(* PLC project Math Expression Evaluator, CODESYS CODESYS V3.5 SP18 Patch 5 *)
(* stored: creationDateTime 2024-02-04T11:49:45.7079355, version 0.1.0.0, modificationDateTime 2024-02-04T11:49:30.3793356, organization GG *)
(* The Math Expression Evaluator evaluates math expressions (terms).

See the documentation folder for an introduction (the folder itself). *)

TYPE typExpressionStep : STRUCT
  atTokens : ARRAY[0..ParameterList.uiMaxExpressionTokens] OF typExpressionToken;
  uiCountTokens : UINT;
  uiInternalVariableTarget : UINT;
END_STRUCT;
END_TYPE

TYPE typExpressionToken : STRUCT
  eType : eTokenType;
  uiGroupNumber : UINT;
  sIdentifier : STRING(5);
  uiArgsCount : UINT;
  xArgsVariable : BOOL;
  lrValue : LREAL;
END_STRUCT;
END_TYPE

TYPE typStepizeGroupFound : STRUCT
  uiTokenIndex : UINT;
  uiGroupNumber : UINT;
  xExpandMore : BOOL;
END_STRUCT;
END_TYPE

TYPE typStepizeRewriteTokenSkips : STRUCT
  uiStart : UINT;
  uiEnd : UINT;
  uiVarNum : UINT;
END_STRUCT;
END_TYPE

(* A division by zero is not allowed and this ENUM describes how such a situation is handled. - ERROR: An error is returned - RESULT_IS_ZERO: The result is simply set to 0.0 and no error is returned - DIVISOR_IS_ONE: The divisor is set to 1.0 instead and the operation is being carried out *)
{attribute 'qualified_only'}
{attribute 'strict'}
TYPE eDivisionByZeroHandling : (ERROR := 0, RESULT_IS_ZERO, DIVISOR_IS_ONE);
END_TYPE

{attribute 'qualified_only'}
{attribute 'strict'}
TYPE eTokenType : (INVALID := 0, NUMBER, VARIABLE, GROUP_START, GROUP_END, MATH_OP, FUNCTION_CALL, FUNCTION_CALL_END, INTERNAL_VAR := 99);
END_TYPE

TYPE typExpressionOperationSteps : STRUCT
  atSteps : ARRAY[0..ParameterList.uiMaxStepsPerOperation] OF typExpressionStep;
  uiCountSteps : UINT;
END_STRUCT;
END_TYPE

TYPE typTokenizedExpression : STRUCT
  atTokens : ARRAY[0..ParameterList.uiMaxExpressionTokens] OF typExpressionToken;
  uiCountTokens : UINT;
END_STRUCT;
END_TYPE

{attribute 'qualified_only'}
VAR_GLOBAL CONSTANT  (* Constants *)
  CHAR_WHITESPACE : BYTE := 32;
  CHAR_NEWLINE : BYTE := 10;
  CHAR_CAR_RETURN : BYTE := 13;
  CHAR_VARIABLE : BYTE := 92;  (* \ *)
  CHAR_GROUP_START : BYTE := 40;  (* ( *)
  CHAR_GROUP_END : BYTE := 41;  (* ) *)
  CHAR_COMMA : BYTE := 44;  (* , *)
  CHAR_DOT : BYTE := 46;  (* . *)
  CHAR_LC_E : BYTE := 101;  (* e *)
  CHAR_ADD : BYTE := 43;  (* + (also used for sign) *)
  CHAR_SUB : BYTE := 45;  (* - (also used for sign) *)
  CHAR_MUL : BYTE := 42;  (* * *)
  CHAR_DIV : BYTE := 47;  (* / *)
  CHAR_EXP : BYTE := 94;  (* ^ *)
  CHAR_MOD : BYTE := 37;  (* % *)
  ASCII_ALPHA_START : BYTE := 65;  (* A *)
  ASCII_ALPHA_END : BYTE := 90;  (* Z *)
  ASCII_NUM_START : BYTE := 48;  (* 0 *)
  ASCII_NUM_END : BYTE := 57;  (* 9 *)
  MAX_FUN_ARGS : UINT := 9;
  FUN_ABS : STRING(5) := 'ABS';  (* Single arg functions *)
  FUN_ACOS : STRING(5) := 'ACOS';
  FUN_ASIN : STRING(5) := 'ASIN';
  FUN_ATAN : STRING(5) := 'ATAN';
  FUN_CEIL : STRING(5) := 'CEIL';
  FUN_COS : STRING(5) := 'COS';
  FUN_DEG : STRING(5) := 'DEG';
  FUN_FLOOR : STRING(5) := 'FLOOR';
  FUN_LOG : STRING(5) := 'LOG';
  FUN_LN : STRING(5) := 'LN';
  FUN_RAD : STRING(5) := 'RAD';
  FUN_ROUND : STRING(5) := 'ROUND';
  FUN_SIN : STRING(5) := 'SIN';
  FUN_SQRT : STRING(5) := 'SQRT';
  FUN_TAN : STRING(5) := 'TAN';
  FUN_TRUNC : STRING(5) := 'TRUNC';  (* Dual arg functions *)
  FUN_LIMIT : STRING(5) := 'LIMIT';  (* Triple arg functions *)
  FUN_AVGA : STRING(5) := 'AVG';  (* Variable arg functions (2..9) *)
  FUN_MAX : STRING(5) := 'MAX';
  FUN_MIN : STRING(5) := 'MIN';
END_VAR

{attribute 'parameterlist'}
{attribute 'qualified_only'}
VAR_GLOBAL CONSTANT  (* ParameterList *)
  uiMaxExpressionTokens : UINT := 63;  (* The maximum amount of tokens to support parsing (compiling) - the counting starts from 0, so add 1 to the number in your mind *)
  uiMaxInternalVars : UINT := 16;  (* The maximum amount of internal variables per expression *)
  uiMaxStepsPerOperation : UINT := 15;  (* The maximum amount of steps per operation - the counting starts from 0, so add 1 to the number in your mind *)
  eDivisionByZero : eDivisionByZeroHandling := eDivisionByZeroHandling.ERROR;  (* Describes how a division by zero situation is to be handled *)
END_VAR

(* Evaluates a function call. First all necessary arguments are resolved to LREAL and then the function gets executed. The return value will indicate a successful evaluation. *)
{attribute 'qualified_only'}
FUNCTION FuEvaluateFunctionCall : BOOL
  VAR_INPUT
    typFunctionToken : typExpressionToken;
    uiMaxCursor : UINT;
    {attribute 'variable_length_array_original_scope' := 'Inout'}
    {attribute 'variable_length_array' := 'ARRAY[*] OF typExpressionToken'}
    {attribute 'Dimensions' := '1'}
    atTokens : POINTER TO typExpressionToken;
  END_VAR
  VAR_IN_OUT
    uiCursor : UINT;
  END_VAR
  VAR_INPUT
    {attribute 'variable_length_array_original_scope' := 'Inout'}
    {attribute 'variable_length_array' := 'ARRAY[*] OF LREAL'}
    {attribute 'Dimensions' := '1'}
    alrVariables : POINTER TO LREAL;
    {attribute 'variable_length_array_original_scope' := 'Inout'}
    {attribute 'variable_length_array' := 'ARRAY[*] OF LREAL'}
    {attribute 'Dimensions' := '1'}
    alrInternalVariables : POINTER TO LREAL;
  END_VAR
  VAR_OUTPUT
    lrResult : LREAL;
    sError : STRING;
  END_VAR
  VAR
    i : UINT;
    j : UINT;
    tempArgs : ARRAY[0..8] OF LREAL;
    tempHelperValue : LREAL;
  END_VAR
  VAR CONSTANT
    CONST_PI : LREAL := 3.14159265359;
  END_VAR

            IF typFunctionToken.eType <> eTokenType.FUNCTION_CALL THEN
    sError := Standard.CONCAT('Invalid function call token at ', TO_STRING(uiCursor));
    RETURN;
END_IF

IF uiCursor + typFunctionToken.uiArgsCount > uiMaxCursor THEN
    sError := Standard.CONCAT('Not enough arguments for function call at ', TO_STRING(uiCursor));
    RETURN;
END_IF

FOR i := 0 TO (typFunctionToken.uiArgsCount - 1) BY 1 DO
    j := uiCursor + i + 1;
    
    IF NOT FuEvaluateTokenSingle(atTokens[j], j, alrVariables, alrInternalVariables, lrResult => tempArgs[i], sError => sError) THEN
        RETURN;
    END_IF
END_FOR

uiCursor := uiCursor + typFunctionToken.uiArgsCount;

IF typFunctionToken.sIdentifier = Constants.FUN_ABS THEN
    FuEvaluateFunctionCall := TRUE;
    lrResult := ABS(tempArgs[0]);
ELSIF typFunctionToken.sIdentifier = Constants.FUN_ACOS THEN
    FuEvaluateFunctionCall := TRUE;
    lrResult := ACOS(tempArgs[0]);
ELSIF typFunctionToken.sIdentifier = Constants.FUN_ASIN THEN
    FuEvaluateFunctionCall := TRUE;
    lrResult := ASIN(tempArgs[0]);
ELSIF typFunctionToken.sIdentifier = Constants.FUN_ATAN THEN
    FuEvaluateFunctionCall := TRUE;
    lrResult := ATAN(tempArgs[0]);
ELSIF typFunctionToken.sIdentifier = Constants.FUN_CEIL THEN
    FuEvaluateFunctionCall := TRUE;
    lrResult := FPU.Ceil(tempArgs[0]);
ELSIF typFunctionToken.sIdentifier = Constants.FUN_COS THEN
    FuEvaluateFunctionCall := TRUE;
    lrResult := COS(tempArgs[0]);
ELSIF typFunctionToken.sIdentifier = Constants.FUN_DEG THEN
    FuEvaluateFunctionCall := TRUE;
    lrResult := tempArgs[0] * 180 / CONST_PI;
ELSIF typFunctionToken.sIdentifier = Constants.FUN_FLOOR THEN
    FuEvaluateFunctionCall := TRUE;
    lrResult := FPU.Floor(tempArgs[0]);
ELSIF typFunctionToken.sIdentifier = Constants.FUN_LOG THEN
    FuEvaluateFunctionCall := TRUE;
    lrResult := LOG(tempArgs[0]);
ELSIF typFunctionToken.sIdentifier = Constants.FUN_LN THEN
    FuEvaluateFunctionCall := TRUE;
    lrResult := LN(tempArgs[0]);
ELSIF typFunctionToken.sIdentifier = Constants.FUN_RAD THEN
    FuEvaluateFunctionCall := TRUE;
    lrResult := tempArgs[0] * CONST_PI / 180;
ELSIF typFunctionToken.sIdentifier = Constants.FUN_ROUND THEN
    FuEvaluateFunctionCall := TRUE;
    
    IF (tempArgs[0] - FPU.Truncate(tempArgs[0])) >= 0.5 THEN
        lrResult := FPU.Ceil(tempArgs[0]);
    ELSE
        lrResult := FPU.Floor(tempArgs[0]);
    END_IF
ELSIF typFunctionToken.sIdentifier = Constants.FUN_SIN THEN
    FuEvaluateFunctionCall := TRUE;
    lrResult := SIN(tempArgs[0]);
ELSIF typFunctionToken.sIdentifier = Constants.FUN_SQRT THEN
    FuEvaluateFunctionCall := TRUE;
    lrResult := SQRT(tempArgs[0]);
ELSIF typFunctionToken.sIdentifier = Constants.FUN_TAN THEN
    FuEvaluateFunctionCall := TRUE;
    lrResult := TAN(tempArgs[0]);
ELSIF typFunctionToken.sIdentifier = Constants.FUN_TRUNC THEN
    FuEvaluateFunctionCall := TRUE;
    
    tempHelperValue := EXPT(10, tempArgs[1]);
    lrResult := FPU.Truncate((tempArgs[0] * tempHelperValue)) / tempHelperValue;
ELSIF typFunctionToken.sIdentifier = Constants.FUN_LIMIT THEN
    FuEvaluateFunctionCall := TRUE;
    lrResult := LIMIT(tempArgs[0], tempArgs[1], tempArgs[2]);
ELSIF typFunctionToken.sIdentifier = Constants.FUN_AVGA THEN
    FuEvaluateFunctionCall := TRUE;
    
    tempHelperValue := 0.0;
    FOR i := 0 TO (typFunctionToken.uiArgsCount - 1) BY 1 DO
        tempHelperValue := tempHelperValue + tempArgs[i];
    END_FOR
    
    lrResult := tempHelperValue / typFunctionToken.uiArgsCount;
ELSIF typFunctionToken.sIdentifier = Constants.FUN_MAX THEN
    FuEvaluateFunctionCall := TRUE;
    
    lrResult := -1.7976931348623157E+308;
    FOR i := 0 TO (typFunctionToken.uiArgsCount - 1) BY 1 DO
        IF tempArgs[i] > lrResult THEN
            lrResult := tempArgs[i];
        END_IF
    END_FOR
ELSIF typFunctionToken.sIdentifier = Constants.FUN_MIN THEN
    FuEvaluateFunctionCall := TRUE;
    
    lrResult := 1.7976931348623157E+308;
    FOR i := 0 TO (typFunctionToken.uiArgsCount - 1) BY 1 DO
        IF tempArgs[i] < lrResult THEN
            lrResult := tempArgs[i];
        END_IF
    END_FOR
ELSE
    sError := Standard.CONCAT('Function not implemented: ', typFunctionToken.sIdentifier);
END_IF

          
END_FUNCTION

(* Evaluates a math operation. First both tokens are resolved to LREAL values and then the selected operation takes place. In general, if any of the operands is a special LREAL value, then an error is returned. For Division (/), division by zero yields into an error (depends on ParameterList setting). For MODULO (%), both tokens are converted to LINT and the result is converted back to LREAL. The return value will indicate a successful evaluation. *)
{attribute 'qualified_only'}
FUNCTION FuEvaluateMathOp : BOOL
  VAR_INPUT
    typOp : typExpressionToken;
    typToken1 : typExpressionToken;
    typToken2 : typExpressionToken;
    uiCursor : UINT;  (* Only for error message *)
    {attribute 'variable_length_array_original_scope' := 'Inout'}
    {attribute 'variable_length_array' := 'ARRAY[*] OF LREAL'}
    {attribute 'Dimensions' := '1'}
    alrVariables : POINTER TO LREAL;
    {attribute 'variable_length_array_original_scope' := 'Inout'}
    {attribute 'variable_length_array' := 'ARRAY[*] OF LREAL'}
    {attribute 'Dimensions' := '1'}
    alrInternalVariables : POINTER TO LREAL;
  END_VAR
  VAR_OUTPUT
    lrResult : LREAL;
    sError : STRING;
  END_VAR
  VAR
    tempOperatorByte : BYTE;
    tempNumber1 : LREAL;
    tempNumber2 : LREAL;
  END_VAR

            IF typOp.eType <> eTokenType.MATH_OP THEN
    sError := Standard.CONCAT('Invalid math operation token at ', TO_STRING(uiCursor));
    RETURN;
END_IF

// Change STRING identifier to BYTE (to match on FuTokenizeExpression strings)
tempOperatorByte := typOp.sIdentifier[0];

// Resolve first token to LREAL
IF NOT FuEvaluateTokenSingle(typToken1, uiCursor, alrVariables, alrInternalVariables, lrResult => tempNumber1, sError => sError) THEN
    FuEvaluateMathOp := FALSE;
    RETURN;
END_IF

// Resolve second token to LREAL
IF NOT FuEvaluateTokenSingle(typToken2, uiCursor, alrVariables, alrInternalVariables, lrResult => tempNumber2, sError => sError) THEN
    FuEvaluateMathOp := FALSE;
    RETURN;
END_IF

IF NOT FPU.IsLRealNumber(tempNumber1) THEN
    FuEvaluateMathOp := FALSE;
    sError := Standard.CONCAT('Special LREAL value is not valid: ', TO_STRING(tempNumber1));
    RETURN;
ELSIF NOT FPU.IsLRealNumber(tempNumber2) THEN
    FuEvaluateMathOp := FALSE;
    sError := Standard.CONCAT('Special LREAL value is not valid: ', TO_STRING(tempNumber2));
    RETURN;
END_IF

IF tempOperatorByte = Constants.CHAR_ADD THEN
    lrResult := tempNumber1 + tempNumber2;
ELSIF tempOperatorByte = Constants.CHAR_SUB THEN
    lrResult := tempNumber1 - tempNumber2;
ELSIF tempOperatorByte = Constants.CHAR_MUL THEN
    lrResult := tempNumber1 * tempNumber2;
ELSIF tempOperatorByte = Constants.CHAR_DIV THEN
    IF tempNumber2 = 0.0 THEN
        CASE ParameterList.eDivisionByZero OF
            eDivisionByZeroHandling.RESULT_IS_ZERO:
                FuEvaluateMathOp := TRUE;
                lrResult := 0.0;
                RETURN;
            
            eDivisionByZeroHandling.DIVISOR_IS_ONE:
                tempNumber2 := 1.0;
        ELSE
            sError := 'Division by zero is not allowed';
            RETURN;
        END_CASE
    END_IF
    
    lrResult := tempNumber1 / tempNumber2;
ELSIF tempOperatorByte = Constants.CHAR_EXP THEN
    lrResult := EXPT(tempNumber1, tempNumber2);
ELSIF tempOperatorByte = Constants.CHAR_MOD THEN
    lrResult := LINT_TO_LREAL((LREAL_TO_LINT(tempNumber1) MOD LREAL_TO_LINT(tempNumber2)));
ELSE
    sError := Standard.CONCAT('Unknown math operator at position ', TO_STRING(uiCursor));
    RETURN;
END_IF

FuEvaluateMathOp := TRUE;

          
END_FUNCTION

(* Evaluates an operation expression. For example "5 + 2", but not "5 + 2 + 1". The return value will indicate a successful evaluation. *)
{attribute 'qualified_only'}
FUNCTION FuEvaluateOperation : BOOL
  VAR_INPUT
    uiMaxCursor : UINT;
    {attribute 'variable_length_array_original_scope' := 'Inout'}
    {attribute 'variable_length_array' := 'ARRAY[*] OF typExpressionToken'}
    {attribute 'Dimensions' := '1'}
    atTokens : POINTER TO typExpressionToken;
  END_VAR
  VAR_IN_OUT
    uiCursor : UINT;
  END_VAR
  VAR_INPUT
    {attribute 'variable_length_array_original_scope' := 'Inout'}
    {attribute 'variable_length_array' := 'ARRAY[*] OF LREAL'}
    {attribute 'Dimensions' := '1'}
    alrVariables : POINTER TO LREAL;
    {attribute 'variable_length_array_original_scope' := 'Inout'}
    {attribute 'variable_length_array' := 'ARRAY[*] OF LREAL'}
    {attribute 'Dimensions' := '1'}
    alrInternalVariables : POINTER TO LREAL;
  END_VAR
  VAR_OUTPUT
    lrResult : LREAL;
    sError : STRING;
  END_VAR
  VAR
    tempLowerBound : UINT;
    tempUpperBound : UINT;
    tempToken1 : typExpressionToken;
    tempToken2 : typExpressionToken;
    tempToken3 : typExpressionToken;
    tempVariableNr : UINT;
  END_VAR

            tempLowerBound := TO_UINT(LOWER_BOUND(atTokens, 1));
tempUpperBound := MIN(uiMaxCursor, TO_UINT(UPPER_BOUND(atTokens, 1)));

tempToken1 := atTokens[uiCursor];

CASE tempToken1.eType OF
    eTokenType.INVALID, eTokenType.MATH_OP, eTokenType.GROUP_START, eTokenType.GROUP_END, eTokenType.FUNCTION_CALL_END:
        sError := Standard.CONCAT('Invalid token at position ', TO_STRING(uiCursor));
        RETURN;
    
    eTokenType.FUNCTION_CALL:
        FuEvaluateOperation := FuEvaluateFunctionCall(
            tempToken1,
            tempUpperBound,
            atTokens,
            uiCursor,
            alrVariables,
            alrInternalVariables,
            lrResult => lrResult,
            sError => sError
        );
        RETURN;
END_CASE

// If we're past the maximum position/cursor, evaluate the token (it should be a variable or number)
IF uiCursor = uiMaxCursor AND_THEN FuEvaluateTokenSingle(tempToken1, uiCursor, alrVariables, alrInternalVariables, lrResult => lrResult, sError => sError) THEN
    RETURN;
END_IF

uiCursor := uiCursor + 1;

// The first token wasn't a variable or number and we're out of bounds, error out
IF uiCursor > tempUpperBound THEN
    sError := 'Array upper bounds violation (not enough tokens)';
    RETURN;
END_IF

tempToken2 := atTokens[uiCursor];

CASE tempToken2.eType OF
    eTokenType.MATH_OP:
        uiCursor := uiCursor + 1;
        IF uiCursor > tempUpperBound THEN
            sError := 'Array upper bounds violation (not enough tokens)';
            RETURN;
        END_IF
        
        FuEvaluateOperation := FuEvaluateMathOp(
            tempToken2,
            tempToken1,
            atTokens[uiCursor],
            uiCursor,
            alrVariables,
            alrInternalVariables,
            lrResult => lrResult,
            sError => sError
        );
        RETURN;
ELSE
    sError := Standard.CONCAT('Invalid token at position ', TO_STRING(uiCursor));
    RETURN;
END_CASE

          
END_FUNCTION

(* Evaluates a single step. For multiple token "expressions" (i.e. "5 + 2 + 1"), the term will be evaluated left to right (in token order). The return value will indicate a successful expression evaluation. *)
{attribute 'qualified_only'}
FUNCTION FuEvaluateStep : BOOL
  VAR_INPUT
    typStep : typExpressionStep;
  END_VAR
  VAR_OUTPUT
    lrResult : LREAL;
    sError : STRING;
  END_VAR
  VAR_INPUT
    {attribute 'variable_length_array_original_scope' := 'Inout'}
    {attribute 'variable_length_array' := 'ARRAY[*] OF LREAL'}
    {attribute 'Dimensions' := '1'}
    alrVariables : POINTER TO LREAL;
    {attribute 'variable_length_array_original_scope' := 'Inout'}
    {attribute 'variable_length_array' := 'ARRAY[*] OF LREAL'}
    {attribute 'Dimensions' := '1'}
    alrInternalVariables : POINTER TO LREAL;
  END_VAR
  VAR
    i : UINT;
    tempMaxCursor : UINT;
    tempResult : LREAL;
    tempError : STRING;
  END_VAR

            IF typStep.uiCountTokens = 0 THEN
    FuEvaluateStep := TRUE;
    RETURN;
END_IF

lrResult := 0.0;
sError := '';

tempMaxCursor := typStep.uiCountTokens - 1;
FOR i := 0 TO tempMaxCursor BY 1 DO
    // For operations like "5 + 3 + 1", we need for the second step "+ 1"
    // to insert the previous result of "5 + 3", so we rewind one and overwrite it
    IF i > 0 AND_THEN typStep.atTokens[i].eType = eTokenType.MATH_OP THEN
        i := i - 1;
        typStep.atTokens[i].eType := eTokenType.NUMBER;
        typStep.atTokens[i].lrValue := tempResult;
    END_IF
    
    IF NOT FuEvaluateOperation(tempMaxCursor, typStep.atTokens, i, alrVariables, alrInternalVariables, lrResult => tempResult, sError => tempError) THEN
        sError := tempError;
        RETURN;
    END_IF
END_FOR

lrResult := tempResult;
FuEvaluateStep := TRUE;

          
END_FUNCTION

(* Evaluates token types that are considered "single". This includes: numbers, variables, internal variables. The return value will indicate a successful evaluation. *)
{attribute 'qualified_only'}
FUNCTION FuEvaluateTokenSingle : BOOL
  VAR_INPUT
    typToken : typExpressionToken;
    uiCursor : UINT;  (* Only for error message *)
    {attribute 'variable_length_array_original_scope' := 'Inout'}
    {attribute 'variable_length_array' := 'ARRAY[*] OF LREAL'}
    {attribute 'Dimensions' := '1'}
    alrVariables : POINTER TO LREAL;
    {attribute 'variable_length_array_original_scope' := 'Inout'}
    {attribute 'variable_length_array' := 'ARRAY[*] OF LREAL'}
    {attribute 'Dimensions' := '1'}
    alrInternalVariables : POINTER TO LREAL;
  END_VAR
  VAR_OUTPUT
    lrResult : LREAL;
    sError : STRING;
  END_VAR
  VAR
    tempVariableNr : UINT;
  END_VAR

            CASE typToken.eType OF
    eTokenType.NUMBER:
        FuEvaluateTokenSingle := TRUE;
        lrResult := typToken.lrValue;
    
    eTokenType.VARIABLE, eTokenType.INTERNAL_VAR:
        FuEvaluateTokenSingle := FuEvaluateVariable(typToken, uiCursor, alrVariables, alrInternalVariables, lrResult => lrResult, sError => sError);
ELSE
    sError := Standard.CONCAT('Invalid single token at position ', TO_STRING(uiCursor));
END_CASE

          
END_FUNCTION

(* Evaluates variables and internal variables to their LREAL value. The return value will indicate a successful evaluation. *)
{attribute 'qualified_only'}
FUNCTION FuEvaluateVariable : BOOL
  VAR_INPUT
    typToken : typExpressionToken;
    uiCursor : UINT;  (* Only for error message *)
    {attribute 'variable_length_array_original_scope' := 'Inout'}
    {attribute 'variable_length_array' := 'ARRAY[*] OF LREAL'}
    {attribute 'Dimensions' := '1'}
    alrVariables : POINTER TO LREAL;
    {attribute 'variable_length_array_original_scope' := 'Inout'}
    {attribute 'variable_length_array' := 'ARRAY[*] OF LREAL'}
    {attribute 'Dimensions' := '1'}
    alrInternalVariables : POINTER TO LREAL;
  END_VAR
  VAR_OUTPUT
    lrResult : LREAL;
    sError : STRING;
  END_VAR
  VAR
    tempVariableNr : UINT;
  END_VAR

            CASE typToken.eType OF
    eTokenType.VARIABLE:
        tempVariableNr := TO_UINT(typToken.lrValue);
        
        IF LOWER_BOUND(alrVariables, 1) <= tempVariableNr AND_THEN tempVariableNr <= UPPER_BOUND(alrVariables, 1) THEN
            FuEvaluateVariable := TRUE;
            lrResult := alrVariables[tempVariableNr];
        ELSE
            sError := Standard.CONCAT('Unknown variable ', TO_STRING(tempVariableNr));
        END_IF
    
    eTokenType.INTERNAL_VAR:
        tempVariableNr := TO_UINT(typToken.lrValue);
        
        IF LOWER_BOUND(alrInternalVariables, 1) <= tempVariableNr AND_THEN tempVariableNr <= UPPER_BOUND(alrInternalVariables, 1) THEN
            FuEvaluateVariable := TRUE;
            lrResult := alrInternalVariables[tempVariableNr];
        ELSE
            sError := Standard.CONCAT('Unknown internal variable ', TO_STRING(tempVariableNr));
        END_IF
ELSE
    sError := Standard.CONCAT('Not a variable token at position ', TO_STRING(uiCursor));
END_CASE

          
END_FUNCTION

(* Slightly modified version of: https://forge.codesys.com/forge/talk/Runtime/thread/6ae1b1ff98/#31a5/f035/66da/5ba5/1553/b75d/ce46 This version uses instead of basic datatypes a struct and sorts it by {group number} and then {token index} *)
{attribute 'qualified_only'}
FUNCTION FuInsertSortStepizeGroupFound : BOOL
  VAR_INPUT
    pbBuffer : POINTER TO BYTE;  (* Pointer to buffer (array) *)
    diElements : DINT;  (* Array length *)
  END_VAR
  VAR
    tempDataSize : UINT;  (* Element size *)
    tempIndex : DINT;  (* Loop index *)
    tempMinIndex : DINT;  (* Loop lowest index tested *)
    tempMaxIndex : DINT;  (* Loop highest index tested *)
    tempCurrentIndex : DINT;  (* Loop current tested element index *)
    tempTemp : ARRAY[1..8] OF BYTE;  (* Store temp value *)
    tempPtrElement1 : POINTER TO typStepizeGroupFound;  (* Pointer operator, current element *)
    tempPtrElement2 : POINTER TO typStepizeGroupFound;  (* Pointer operator, insert element *)
    tempElement1 : typStepizeGroupFound;
    tempElement2 : typStepizeGroupFound;
  END_VAR

            tempDataSize := SIZEOF(typStepizeGroupFound);

FOR tempIndex := 1 TO diElements - 1 DO
    // Highest index tested
    tempMaxIndex := tempIndex;
    
    // Lowest index tested
    tempMinIndex := -1;
    
    // Element we need to insert
    tempPtrElement2 := pbBuffer + TO_UDINT(tempDataSize*tempIndex);
    
    REPEAT
        // Current test index
        tempCurrentIndex := tempMinIndex + (tempMaxIndex - tempMinIndex) / 2;
        
        // Get element at current test index
        tempPtrElement1 := pbBuffer + TO_UDINT(tempDataSize*tempCurrentIndex);
        
        // Test for ordering
        SysMem.SysMemCpy(pDest := ADR(tempElement1), pSrc := tempPtrElement1, udiCount := tempDataSize);
        SysMem.SysMemCpy(pDest := ADR(tempElement2), pSrc := tempPtrElement2, udiCount := tempDataSize);
        
        IF tempElement1.uiGroupNumber = tempElement2.uiGroupNumber THEN
            IF tempElement1.uiTokenIndex > tempElement2.uiTokenIndex THEN
                tempMaxIndex := tempCurrentIndex;
            ELSE
                tempMinIndex := tempCurrentIndex;
            END_IF
        ELSIF tempElement1.uiGroupNumber > tempElement2.uiGroupNumber THEN
            tempMaxIndex := tempCurrentIndex;
        ELSE
            tempMinIndex := tempCurrentIndex;
        END_IF
    UNTIL
        (tempMaxIndex - tempMinIndex) < 2
    END_REPEAT
    
    // Save value to insert
    SysMem.SysMemCpy(pDest := ADR(tempTemp), pSrc := tempPtrElement2, udiCount := tempDataSize);
    
    // Move block
    SysMem.SysMemMove(
        pDest := (pbBuffer + tempDataSize * (TO_UDINT(tempMaxIndex) + 1)),
        pSrc := (pbBuffer + TO_UDINT((tempDataSize * tempMaxIndex))),
        udiCount := (tempDataSize * TO_UDINT(tempIndex - tempMaxIndex))
    );
    
    // set key
    SysMem.SysMemCpy(pDest := (pbBuffer + tempDataSize * TO_UDINT(tempMaxIndex)), pSrc := ADR(tempTemp), udiCount := tempDataSize);
END_FOR

FuInsertSortStepizeGroupFound := TRUE;

          
END_FUNCTION

(* This is a high level Math Expression Evaluator. It uses the low level functions to build a high level API. As such it combines the three fundamental low level functions. All expressions use LREAL as data type for operations, which is also the result output. The following math operation behaviour applies: - In general: If any of the operands is a special value (+Inf, -Inf, NaN), then an error is returned - For Division (/): Division by zero yields depending on ParameterList.eDivisionByZero into an error or not - For Modulo (%): Both operands are converted to LINT and the result is converted back to LREAL Once evaluation gets triggered, the first time it gets triggered (or on expression change) it will tokenize and "stepize" the given expression. Once these steps pass successfully, it will evaluate the expressions. These output will change state accordingly. This function block will reset the "xTrigger" IN_OUT variable once it's done. Since all the necessary low level functions are synchronous, execution of this function block is also synchronous and thus xTrigger will get reset immediately after execution. *)
{attribute 'qualified_only'}
FUNCTION_BLOCK FbMathExpressionEvaluator
  VAR_INPUT
    sExpression : STRING(255);  (* The expression string to tokenize *)
  END_VAR
  VAR_OUTPUT
    xDone : BOOL;  (* Evaluation is done (either successfully or not) - set for one cycle *)
    xError : BOOL;  (* Error during any of the evaluator steps *)
    sError : STRING;  (* Error message (may also contain nonsense if function returns TRUE) *)
    lrResult : LREAL;  (* Result output *)
  END_VAR
  VAR_IN_OUT
    xTrigger : BOOL;  (* Trigger evaluation, gets automatically reset *)
  END_VAR
  VAR_INPUT
    {attribute 'variable_length_array_original_scope' := 'Inout'}
    {attribute 'variable_length_array' := 'ARRAY[*] OF LREAL'}
    {attribute 'Dimensions' := '1'}
    alrVariables : POINTER TO LREAL;  (* Variables to use *)
  END_VAR
  VAR
    staticUsedExpression : STRING(255);
    staticSteppedExpression : typExpressionOperationSteps;
  END_VAR
  VAR_TEMP
    tempSuccess : BOOL;
    tempTokenizedExpression : typTokenizedExpression;
  END_VAR

            IF xTrigger THEN
    IF sExpression = '' THEN
        xTrigger := FALSE;
        xDone := TRUE;
        xError := TRUE;
        sError := 'Empty expression';
        lrResult := 0.0;
        RETURN;
    END_IF
    
    IF staticUsedExpression <> sExpression THEN
        staticUsedExpression := '';
        
        tempSuccess := FuTokenizeExpression(sExpression, typExpression => tempTokenizedExpression, sError => sError);
        IF NOT tempSuccess THEN
            xTrigger := FALSE;
            xDone := TRUE;
            xError := TRUE;
            lrResult := 0.0;
            RETURN;
        END_IF
        
        sError := '';
        
        tempSuccess := FuStepizeExpression(tempTokenizedExpression, typSteps => staticSteppedExpression);
        IF NOT tempSuccess THEN
            xTrigger := FALSE;
            xDone := TRUE;
            xError := TRUE;
            sError := 'Error during stepize';
            lrResult := 0.0;
            RETURN;
        END_IF
        
        staticUsedExpression := sExpression;
    END_IF
    
    IF FuEvaluateExpression(staticSteppedExpression, alrVariables, lrResult => lrResult, sError => sError) THEN
        // Assert error string is empty if no error
        sError := '';
    ELSE
        xError := TRUE;
    END_IF
    
    xTrigger := FALSE;
    xDone := TRUE;
    
    RETURN;
END_IF

xDone := FALSE;

          
END_FUNCTION_BLOCK

(* Evaluates the expression. All expressions use LREAL as data type for operations, which is also the result output. The following math operation behaviour applies: - In general: If any of the operands is a special value (+Inf, -Inf, NaN), then an error is returned - For Division (/): Division by zero yields depending on ParameterList.eDivisionByZero into an error or not - For Modulo (%): Both operands are converted to LINT and the result is converted back to LREAL The return value will indicate a successful evaluation. *)
{attribute 'qualified_only'}
FUNCTION FuEvaluateExpression : BOOL
  VAR_INPUT
    typExpressionSteps : typExpressionOperationSteps;  (* The expression providing steps for complex terms *)
    {attribute 'variable_length_array_original_scope' := 'Input'}
    {attribute 'variable_length_array' := 'ARRAY[*] OF LREAL'}
    {attribute 'Dimensions' := '1'}
    alrVariables : POINTER TO LREAL;  (* Variables to use *)
  END_VAR
  VAR_OUTPUT
    lrResult : LREAL;  (* Result output *)
    sError : STRING;  (* Error message *)
  END_VAR
  VAR
    i : UINT;
    tempResult : LREAL;
    tempError : STRING;
    tempInternalVariables : ARRAY[0..ParameterList.uiMaxInternalVars] OF LREAL;
  END_VAR

            IF typExpressionSteps.uiCountSteps = 0 THEN
    FuEvaluateExpression := TRUE;
    RETURN;
END_IF

FOR i := 0 TO (typExpressionSteps.uiCountSteps - 1) BY 1 DO
    IF NOT FuEvaluateStep(typExpressionSteps.atSteps[i],  alrVariables, tempInternalVariables, lrResult => tempResult, sError => tempError) THEN
        sError := tempError;
        RETURN;
    END_IF
    
    // Always have the result in internal variable 0
    tempInternalVariables[0] := tempResult;
    
    IF
        typExpressionSteps.atSteps[i].uiInternalVariableTarget > 0 AND_THEN
        typExpressionSteps.atSteps[i].uiInternalVariableTarget >= 1 AND_THEN
        typExpressionSteps.atSteps[i].uiInternalVariableTarget <= ParameterList.uiMaxInternalVars
    THEN
        tempInternalVariables[typExpressionSteps.atSteps[i].uiInternalVariableTarget] := tempResult;
    END_IF
END_FOR

lrResult := tempResult;
FuEvaluateExpression := TRUE;

          
END_FUNCTION

(* Turns a tokenized expression into a stepized expression, providing steps for each "group" operation to be done, including taking care of ordering. Group operations include function calls and expressions inside (). Operations such as "1 + 5 - 2" are not split up and are evaluated left to right from the evaluator. The return value signifies whether the operation has been successfully completed. This function should only return false, when we run out of internal variables or there are no tokens. *)
{attribute 'qualified_only'}
FUNCTION FuStepizeExpression : BOOL
  VAR_INPUT
    typTokenExpression : typTokenizedExpression;
  END_VAR
  VAR_OUTPUT
    typSteps : typExpressionOperationSteps;
  END_VAR
  VAR
    i : UINT;
    j : UINT;
    tempEndTokenIndex : UINT;
    tempFoundGroups : ARRAY[0..ParameterList.uiMaxExpressionTokens] OF typStepizeGroupFound;  (* Data used throughout each loop iteration *)
    tempCountFoundGroups : UINT;
    tempFoundGroupsTokens : ARRAY[0..ParameterList.uiMaxExpressionTokens] OF typExpressionToken;
    tempCountFoundGroupsTokens : UINT;
    tempLastStartedGroups : ARRAY[0..ParameterList.uiMaxExpressionTokens] OF UINT;
    tempCountLastStartedGroups : UINT;
  END_VAR
  VAR CONSTANT
    {attribute 'suppress_warning_0' := 'C0228'}
    INVALID_TOKEN : typExpressionToken := (eType := eTokenType.INVALID);
    {attribute 'suppress_warning_0' := 'C0228'}
    EMPTY_TOKEN_ARR : ARRAY[0..ParameterList.uiMaxExpressionTokens] OF typExpressionToken;
  END_VAR

            IF typTokenExpression.uiCountTokens = 0 THEN
    RETURN;
END_IF

// Step 1: Find each group and make a list out of it
FOR i := 0 TO (typTokenExpression.uiCountTokens - 1) BY 1 DO
    IF
        typTokenExpression.atTokens[i].eType = eTokenType.GROUP_START OR_ELSE
        typTokenExpression.atTokens[i].eType = eTokenType.FUNCTION_CALL
    THEN
        tempFoundGroups[tempCountFoundGroups].uiTokenIndex := i;
        tempFoundGroups[tempCountFoundGroups].uiGroupNumber := typTokenExpression.atTokens[i].uiGroupNumber;
        
        tempCountFoundGroups := tempCountFoundGroups + 1;
    END_IF
END_FOR

// Skip step 2 and 3 if we found NO groups
IF tempCountFoundGroups > 0 THEN
    // Step 2: Sort the found groups array by group number and then token index
    FuInsertSortStepizeGroupFound(ADR(tempFoundGroups), tempCountFoundGroups);
    
    // Step 3: Consume found groups, take the tokens and insert ASSIGN_INTERNAL_VAR tokens
    //         -> Note: The found groups index + 1 corresponds to the internal variable number
    FOR i := 0 TO (tempCountFoundGroups - 1) BY 1 DO
        tempFoundGroupsTokens := EMPTY_TOKEN_ARR;
        tempCountFoundGroupsTokens := 0;
        
        tempCountLastStartedGroups := 0;
        tempEndTokenIndex := 0;
        
        FOR j := tempFoundGroups[i].uiTokenIndex TO (typTokenExpression.uiCountTokens - 1) BY 1 DO
            IF typTokenExpression.atTokens[j].eType = eTokenType.INVALID THEN
                CONTINUE;
            END_IF
            
            IF typTokenExpression.atTokens[j].eType = eTokenType.GROUP_START AND_THEN typTokenExpression.atTokens[j].uiGroupNumber <> tempFoundGroups[i].uiGroupNumber THEN
                // Another group started, we need to ignore those tokens now
                tempLastStartedGroups[tempCountLastStartedGroups] := typTokenExpression.atTokens[j].uiGroupNumber;
                tempCountLastStartedGroups := tempCountLastStartedGroups + 1;
                
                CONTINUE;
            ELSIF
                typTokenExpression.atTokens[j].eType = eTokenType.GROUP_END AND_THEN
                tempCountLastStartedGroups > 0 AND_THEN
                typTokenExpression.atTokens[j].uiGroupNumber = tempLastStartedGroups[(tempCountLastStartedGroups - 1)]
            THEN
                // Another group ended, we can now start caring again, if the count drops to 0
                tempCountLastStartedGroups := tempCountLastStartedGroups - 1;
                
                CONTINUE; // Taking care of using the internal variable of each group will be done later using "tempSkipTokenHints"
            ELSIF tempCountLastStartedGroups > 0 THEN
                // As long as another group are still open, prevent the other two clauses (the elsif and else) from being able to execute
                CONTINUE;
            END_IF
            
            IF typTokenExpression.atTokens[j].eType = eTokenType.GROUP_END AND_THEN typTokenExpression.atTokens[j].uiGroupNumber = tempFoundGroups[i].uiGroupNumber THEN
                // We've reached the end of our group, stop taking tokens away, add a hint for later about skipping tokens, and exit this loop
                tempEndTokenIndex := j;
                EXIT;
            ELSIF typTokenExpression.atTokens[j].eType = eTokenType.GROUP_START AND_THEN typTokenExpression.atTokens[j].uiGroupNumber = tempFoundGroups[i].uiGroupNumber THEN
                // Ignore group starts of ourself (we dont need those tokens)
                CONTINUE;
            END_IF
            
            IF typTokenExpression.atTokens[j].eType = eTokenType.FUNCTION_CALL_END AND_THEN typTokenExpression.atTokens[j].uiGroupNumber = tempFoundGroups[i].uiGroupNumber THEN
                // We've reached the end of our group, stop taking tokens away, add a hint for later about skipping tokens, and exit this loop
                tempEndTokenIndex := j;
                EXIT;
            END_IF
            
            tempFoundGroupsTokens[tempCountFoundGroupsTokens] := typTokenExpression.atTokens[j];
            tempCountFoundGroupsTokens := tempCountFoundGroupsTokens + 1;
        END_FOR
        
        typSteps.atSteps[typSteps.uiCountSteps].atTokens := tempFoundGroupsTokens;
        typSteps.atSteps[typSteps.uiCountSteps].uiCountTokens := tempCountFoundGroupsTokens;
        typSteps.atSteps[typSteps.uiCountSteps].uiInternalVariableTarget := i + 1;
        
        IF i >= ParameterList.uiMaxInternalVars THEN
            FuStepizeExpression := FALSE;
            RETURN;
        END_IF
        
        // Replace all tokens with invalid tokens, if necessary, the first token will be replaced with INTERNAL_VAR
        FOR j := tempFoundGroups[i].uiTokenIndex TO tempEndTokenIndex BY 1 DO
            typTokenExpression.atTokens[j] := INVALID_TOKEN;
        END_FOR
        
        IF tempFoundGroups[i].uiTokenIndex = 0 AND_THEN tempEndTokenIndex = (typTokenExpression.uiCountTokens - 1) THEN
            ;// Do not generate internal var token, because all tokens are covered
        ELSE
            // Rewrite tokens and replace them with one INTERNAL_VAR and INVALID tokens
            typTokenExpression.atTokens[tempFoundGroups[i].uiTokenIndex] := INVALID_TOKEN;
            typTokenExpression.atTokens[tempFoundGroups[i].uiTokenIndex].eType := eTokenType.INTERNAL_VAR;
            typTokenExpression.atTokens[tempFoundGroups[i].uiTokenIndex].lrValue := TO_LREAL((i + 1));
        END_IF
        
        typSteps.uiCountSteps := typSteps.uiCountSteps + 1;
    END_FOR
END_IF

// Step 4: Rewrite the tokens, skip INVALID tokens
FOR i := 0 TO (typTokenExpression.uiCountTokens - 1) BY 1 DO
    IF typTokenExpression.atTokens[i].eType = eTokenType.INVALID THEN
        CONTINUE;
    END_IF
    
    j := typSteps.atSteps[typSteps.uiCountSteps].uiCountTokens;
    
    typSteps.atSteps[typSteps.uiCountSteps].atTokens[j] := typTokenExpression.atTokens[i];
    typSteps.atSteps[typSteps.uiCountSteps].uiCountTokens := j + 1;
END_FOR

IF typSteps.atSteps[typSteps.uiCountSteps].uiCountTokens > 0 THEN
    typSteps.uiCountSteps := typSteps.uiCountSteps + 1;
END_IF

// Step 5: Profit, each step should now contain a particular operation set
// Note: Operations as "1 + 5 + 6" are handled inline in the evaluator, since the result of the previous op "1 + 5" can be used as "$result + 5"
FuStepizeExpression := TRUE;

          
END_FUNCTION

(* Tokenizes a given math expression into a stream of tokens. The return value signifies whether tokenization was successful, or during tokenization an invalid expression was encountered. Please note, during tokenization not all error cases are checked. *)
{attribute 'qualified_only'}
FUNCTION FuTokenizeExpression : BOOL
  VAR_INPUT
    sExpression : STRING(255);  (* The expression string to tokenize *)
  END_VAR
  VAR_OUTPUT
    typExpression : typTokenizedExpression;  (* The tokenized expression *)
    sError : STRING;  (* Error message *)
  END_VAR
  VAR
    i : UINT;
    j : UINT;
    tempChar : BYTE;
    tempNextChar : BYTE;
    tempFunEndDetected : BOOL;
    tempIndex : UINT;  (* Data used throughout each loop iteration *)
    tempIdentifierStr : STRING(5);
    tempPtrByte : POINTER TO BYTE;
    tempVarOpen : BOOL;
    tempGroupOpen : INT := 0;
    tempGroupNum : UINT := 50;
    tempFunOpen : BOOL;
    tempFunIndex : UINT;
    tempFunArgsCount : UINT;
    tempNumOpen : BOOL;
    tempNumSign : BOOL;  (* TRUE = negative *)
    tempValueStr : STRING(80);
  END_VAR

            IF sExpression = '' THEN
    sError := 'Empty expression';
    RETURN;
END_IF

sError := '';

// Assert a clean string (CODESYS does not assert that the whole string contains NUL bytes, only sets the first byte as NUL byte!)
// tempValueStr is VAR_TEMP and should get completely initialized as an empty string (all bytes = NUL), but the truth is the memory space
// gets reused and thus leftovers from the previous execution can be left there, since only the first byte is set to NUL
// (which is described by CODESYS as "new initialization", which is technically wrong!)
FOR i := 0 TO SIZEOF(tempValueStr) BY 1 DO
    tempValueStr[i] := 0;
END_FOR

FOR i := 0 TO 255 BY 1 DO
    IF sExpression[i] = 0 THEN
        EXIT;
    ELSIF tempIndex > ParameterList.uiMaxExpressionTokens THEN
        sError := 'Too many expressions';
        EXIT;
    END_IF
    
    tempFunEndDetected := FALSE;
    tempIdentifierStr := '';
    tempPtrByte := 0;
    
    tempChar := sExpression[i];
    
    CASE tempChar OF
        Constants.CHAR_WHITESPACE, Constants.CHAR_NEWLINE, Constants.CHAR_CAR_RETURN:
            IF tempNumOpen THEN
                typExpression.atTokens[tempIndex].eType := eTokenType.NUMBER;
                typExpression.atTokens[tempIndex].lrValue := STRING_TO_LREAL(tempValueStr);
                
                tempValueStr := '';
                tempNumOpen := FALSE;
            ELSIF tempVarOpen THEN
                typExpression.atTokens[tempIndex].eType := eTokenType.VARIABLE;
                typExpression.atTokens[tempIndex].lrValue := STRING_TO_LREAL(tempValueStr);
                
                tempValueStr := '';
                tempVarOpen := FALSE;
            ELSE
                CONTINUE; // Ignore whitespace, newline (\n) and carriage return (\r)
            END_IF
        
        Constants.CHAR_VARIABLE:
            IF tempVarOpen OR_ELSE tempNumOpen THEN
                sError := Standard.CONCAT('Unexpected VARIABLE "\" start at token ', TO_STRING(i));
                RETURN;
            END_IF
            
            tempVarOpen := TRUE;
            tempValueStr := '';
            
            CONTINUE;
        
        Constants.CHAR_GROUP_START:
            tempGroupOpen := tempGroupOpen + 1;
            tempGroupNum := tempGroupNum - 1;
            
            typExpression.atTokens[tempIndex].eType := eTokenType.GROUP_START;
            typExpression.atTokens[tempIndex].uiGroupNumber := tempGroupNum;
        
        Constants.CHAR_GROUP_END:
            tempFunEndDetected := (tempFunOpen AND_THEN tempGroupNum = typExpression.atTokens[tempFunIndex].uiGroupNumber);
            
            IF tempNumOpen OR_ELSE tempVarOpen THEN
                typExpression.atTokens[tempIndex].eType := SEL(tempVarOpen, eTokenType.NUMBER, eTokenType.VARIABLE);
                typExpression.atTokens[tempIndex].lrValue := STRING_TO_LREAL(tempValueStr);
                
                tempValueStr := '';
                tempNumOpen := FALSE;
                tempVarOpen := FALSE;
                
                tempIndex := tempIndex + 1;
                typExpression.uiCountTokens := tempIndex;
                
                IF tempFunEndDetected THEN
                    tempFunArgsCount := tempFunArgsCount + 1;
                END_IF
            END_IF
            
            typExpression.atTokens[tempIndex].eType := SEL(tempFunEndDetected, eTokenType.GROUP_END, eTokenType.FUNCTION_CALL_END);
            typExpression.atTokens[tempIndex].uiGroupNumber := tempGroupNum;
            tempGroupNum := tempGroupNum + 1;
            
            IF tempFunEndDetected THEN
                // Assert for variable args functions, we have at least that many arguments,
                // or for fixed args functions, we have that many arguments as currently stored
                IF typExpression.atTokens[tempFunIndex].xArgsVariable THEN
                    IF typExpression.atTokens[tempFunIndex].uiArgsCount > tempFunArgsCount THEN
                        sError := Standard.CONCAT('Not enough arguments for variable function ', typExpression.atTokens[tempFunIndex].sIdentifier);
                        sError := Standard.CONCAT(sError, ', expected: ');
                        sError := Standard.CONCAT(sError, TO_STRING(typExpression.atTokens[tempFunIndex].uiArgsCount));
                        sError := Standard.CONCAT(sError, ', got: ');
                        sError := Standard.CONCAT(sError, TO_STRING(tempFunArgsCount));
                        RETURN;
                    END_IF
                ELSIF typExpression.atTokens[tempFunIndex].uiArgsCount <> tempFunArgsCount THEN
                    sError := Standard.CONCAT('Mismatch arguments count for function ', typExpression.atTokens[tempFunIndex].sIdentifier);
                    sError := Standard.CONCAT(sError, ', expected: ');
                    sError := Standard.CONCAT(sError, TO_STRING(typExpression.atTokens[tempFunIndex].uiArgsCount));
                    sError := Standard.CONCAT(sError, ', got: ');
                    sError := Standard.CONCAT(sError, TO_STRING(tempFunArgsCount));
                    RETURN;
                END_IF
                
                IF tempFunArgsCount > Constants.MAX_FUN_ARGS THEN
                    sError := Standard.CONCAT('Too many function arguments (more than ', TO_STRING(Constants.MAX_FUN_ARGS));
                    sError := Standard.CONCAT(sError, ')');
                    RETURN;
                END_IF
                
                typExpression.atTokens[tempFunIndex].uiArgsCount := tempFunArgsCount;
                
                tempFunOpen := FALSE;
                tempFunArgsCount := 0;
            ELSE
                tempGroupOpen := tempGroupOpen - 1;
            END_IF
        
        Constants.CHAR_COMMA:
            IF NOT tempFunOpen THEN
                sError := Standard.CONCAT('Unexpected COMMA "," outside of function at token ', TO_STRING(i));
                RETURN;
            ELSIF tempNumOpen OR_ELSE tempVarOpen THEN
                typExpression.atTokens[tempIndex].eType := SEL(tempVarOpen, eTokenType.NUMBER, eTokenType.VARIABLE);
                typExpression.atTokens[tempIndex].lrValue := STRING_TO_LREAL(tempValueStr);
                
                tempValueStr := '';
                tempNumOpen := FALSE;
                tempVarOpen := FALSE;
                
                tempIndex := tempIndex + 1;
                typExpression.uiCountTokens := tempIndex;
            END_IF
            
            tempFunArgsCount := tempFunArgsCount + 1;
            CONTINUE;
        
        Constants.CHAR_DOT:
            IF NOT tempNumOpen THEN
                sError := Standard.CONCAT('Unexpected DOT "." outside of number at token ', TO_STRING(i));
                RETURN;
            END_IF
            
            tempValueStr := Standard.CONCAT(tempValueStr, '.');
            CONTINUE;
        
        // "-" must be handled differently, as we may need to handle it as a sign
       Constants. CHAR_ADD, Constants.CHAR_SUB, Constants.CHAR_MUL,
        Constants.CHAR_DIV, Constants.CHAR_EXP, Constants.CHAR_MOD:
            IF tempNumOpen OR_ELSE tempVarOpen THEN
                typExpression.atTokens[tempIndex].eType := SEL(tempVarOpen, eTokenType.NUMBER, eTokenType.VARIABLE);
                typExpression.atTokens[tempIndex].lrValue := STRING_TO_LREAL(tempValueStr);
                
                tempValueStr := '';
                tempNumOpen := FALSE;
                tempVarOpen := FALSE;
                
                tempIndex := tempIndex + 1;
                typExpression.uiCountTokens := tempIndex;
            END_IF
            
            // If operator is ADD/SUB, then peek ahead to see if a number follows immediately (it's a negative number and not an operation)
            tempNextChar := sExpression[(i + 1)];
            IF
                (tempChar = Constants.CHAR_ADD OR_ELSE tempChar = Constants.CHAR_SUB) AND_THEN
                tempNextChar >= Constants.ASCII_NUM_START AND_THEN
                tempNextChar <= Constants.ASCII_NUM_END
            THEN
                tempNumOpen := TRUE;
                tempValueStr := SEL(tempChar = Constants.CHAR_ADD, '-', '');
                
                CONTINUE;
            END_IF
            
            typExpression.atTokens[tempIndex].eType := eTokenType.MATH_OP;
            typExpression.atTokens[tempIndex].sIdentifier := Util.WORD_AS_STRING(tempChar, TRUE);
    ELSE
        IF tempChar >= Constants.ASCII_NUM_START AND_THEN tempChar <= Constants.ASCII_NUM_END THEN
            IF NOT tempVarOpen AND_THEN NOT tempNumOpen THEN
                tempNumOpen := TRUE;
                tempValueStr := '';
            END_IF
            
            tempValueStr := Standard.CONCAT(tempValueStr, TO_STRING((tempChar - Constants.ASCII_NUM_START)));
            CONTINUE;
        ELSIF tempChar >= Constants.ASCII_ALPHA_START AND_THEN tempChar <= Constants.ASCII_ALPHA_END THEN
            // We can not call a function inside a function
            IF tempFunOpen THEN
                sError := Standard.CONCAT('Nested function calls are not supported, found at token ', TO_STRING(i));
                RETURN;
            END_IF
            
            FOR j := i TO (i + 5) BY 1 DO
                IF sExpression[j] = Constants.CHAR_GROUP_START THEN
                    EXIT;
                END_IF
                
                tempIdentifierStr[(j - i)] := sExpression[j];
                
                // Assert string is correctly NUL terminated (prevent "MAXIN" when first "LIMIT" and then "MAX" was tokenized)
                tempIdentifierStr[(j - i + 1)] := 0;
            END_FOR
            
            i := j - 1;
            
            IF
                tempIdentifierStr = Constants.FUN_ABS OR_ELSE
                tempIdentifierStr = Constants.FUN_ACOS OR_ELSE
                tempIdentifierStr = Constants.FUN_ASIN OR_ELSE
                tempIdentifierStr = Constants.FUN_ATAN OR_ELSE
                tempIdentifierStr = Constants.FUN_CEIL OR_ELSE
                tempIdentifierStr = Constants.FUN_COS OR_ELSE
                tempIdentifierStr = Constants.FUN_DEG OR_ELSE
                tempIdentifierStr = Constants.FUN_FLOOR OR_ELSE
                tempIdentifierStr = Constants.FUN_LOG OR_ELSE
                tempIdentifierStr = Constants.FUN_LN OR_ELSE
                tempIdentifierStr = Constants.FUN_RAD OR_ELSE
                tempIdentifierStr = Constants.FUN_ROUND OR_ELSE
                tempIdentifierStr = Constants.FUN_SIN OR_ELSE
                tempIdentifierStr = Constants.FUN_SQRT OR_ELSE
                tempIdentifierStr = Constants.FUN_TAN
            THEN
                // Single arg functions
                typExpression.atTokens[tempIndex].uiArgsCount := 1;
            ELSIF
                tempIdentifierStr = Constants.FUN_TRUNC
            THEN
                // Dual arg functions
                typExpression.atTokens[tempIndex].uiArgsCount := 2;
            ELSIF
                tempIdentifierStr = Constants.FUN_LIMIT
            THEN
                // Triple arg functions
                typExpression.atTokens[tempIndex].uiArgsCount := 3;
            ELSIF
                tempIdentifierStr = Constants.FUN_AVGA OR_ELSE
                tempIdentifierStr = Constants.FUN_MAX OR_ELSE
                tempIdentifierStr = Constants.FUN_MIN
            THEN
                // Variable arg functions (at least 2)
                typExpression.atTokens[tempIndex].uiArgsCount := 2;
                typExpression.atTokens[tempIndex].xArgsVariable := TRUE;
            ELSE
                // Invalid function name
                sError := Standard.CONCAT('Unknown function ', tempIdentifierStr);
                RETURN;
            END_IF
            
            // Peek at the next expression token and check if it's a GROUP_START token
            IF sExpression[(i + 1)] <> Constants.CHAR_GROUP_START THEN
                // If not, invalid expression
                sError := Standard.CONCAT('Expected GROUP_START "(" for function call at token ', TO_STRING((i + 1)));
                RETURN;
            END_IF
            
            // Skip next token, as we've already consumed it
            i := i + 1;
            
            tempFunIndex := tempIndex;
            tempGroupNum := tempGroupNum - 1;
            
            typExpression.atTokens[tempIndex].eType := eTokenType.FUNCTION_CALL;
            typExpression.atTokens[tempIndex].sIdentifier := tempIdentifierStr;
            typExpression.atTokens[tempIndex].uiGroupNumber := tempGroupNum;
            
            tempFunOpen := TRUE;
            tempFunArgsCount := 0;
        ELSE
            // Invalid expression
            sError := Standard.CONCAT('Invalid character at token ', TO_STRING(i));
            RETURN;
        END_IF
    END_CASE
    
    tempIndex := tempIndex + 1;
    typExpression.uiCountTokens := tempIndex;
END_FOR

// If var or num open, close it and append as token
IF tempVarOpen THEN
    typExpression.atTokens[tempIndex].eType := eTokenType.VARIABLE;
    typExpression.atTokens[tempIndex].lrValue := STRING_TO_LREAL(tempValueStr);
    
    tempIndex := tempIndex + 1;
ELSIF tempNumOpen THEN
    typExpression.atTokens[tempIndex].eType := eTokenType.NUMBER;
    typExpression.atTokens[tempIndex].lrValue := STRING_TO_LREAL(tempValueStr);
    
    tempIndex := tempIndex + 1;
END_IF

typExpression.uiCountTokens := tempIndex;
FuTokenizeExpression := (tempIndex > 0 AND_THEN NOT tempVarOpen AND_THEN tempGroupOpen = 0 AND_THEN NOT tempFunOpen);

          
END_FUNCTION
